(* IEC 61131-3 sources: eCockpitGit/test_project/src/%F%00 Library/%F%Structured Buffer Read Write Base/%ITF%ITF_StructWriterBase/%F%Writing, 9 files *)

(* ---- %METH%writeBool.st ---- *)
//This method writes a bool value to the buffer
METHOD writeBool
VAR_INPUT
	value			:BOOL;				//Address of string for the filler text
END_VAR
(*%!%__DELIMITER__%!%*)

(* ---- %METH%writeDint.st ---- *)
//This method writes a dint value to the buffer
METHOD writeDint
VAR_INPUT
	value			:DINT;
END_VAR
(*%!%__DELIMITER__%!%*)

(* ---- %METH%writeDword.st ---- *)
//This method writes a dint value to the buffer
METHOD writeDword
VAR_INPUT
	value			:DWORD;
END_VAR
(*%!%__DELIMITER__%!%*)

(* ---- %METH%writeLint.st ---- *)
//This method writes a dint value to the buffer
METHOD writeLint
VAR_INPUT
	value			:LINT;
END_VAR
(*%!%__DELIMITER__%!%*)

(* ---- %METH%writeLword.st ---- *)
//This method writes a dint value to the buffer
METHOD writeLword
VAR_INPUT
	value			:LWORD;
END_VAR
(*%!%__DELIMITER__%!%*)

(* ---- %METH%writeRaw.st ---- *)
//This method writes a string of any size to the buffer as raw data without qoutes and escape characters
//Should only be used for copying data
METHOD writeRaw
VAR_INPUT
	value			:POINTER TO EASCII;	//Address of string for the filler text
END_VAR
(*%!%__DELIMITER__%!%*)

(* ---- %METH%writeRawLen.st ---- *)
//This method writes a string of a fixed size to the buffer as raw data without qoutes and escape characters
//Should only be used for copying data
// |**Version**|**Author**| **Date** |**Changes**
// | 1         | NSN      | 13-10-21 | Creation
METHOD writeRawLen
VAR_INPUT
	value			:POINTER TO EASCII;	//Address of string for the buffer
	len				:DWORD;				//Amount of bytes to write
END_VAR
(*%!%__DELIMITER__%!%*)

(* ---- %METH%writeReal.st ---- *)
//This method writes a real value to the buffer
METHOD writeReal
VAR_INPUT
	value			:REAL;
END_VAR
(*%!%__DELIMITER__%!%*)

(* ---- %METH%writeString.st ---- *)
//This method writes a string of any size to the buffer
METHOD writeString
VAR_INPUT
	value			:POINTER TO EASCII;	//Address of string for the filler text
END_VAR
(*%!%__DELIMITER__%!%*)
